# B&R Automation Studio project TD52 (part 138)

#### perm_par.var
```iecst
VAR
	pm_Error : UINT; (* permanent value error *) (* Deleted: pm : ParaMem_typ; permanent memory tags mathias, 22.8.11*)
	write_once : BOOL; (* write permanent memory once *)
	pm_len : UDINT; (* permanent value lenght *)
	ModuleName : STRING[35]; (* module name of object *)
	DatObjInfo_01 : DatObjInfo; (* data object info *)
	pm_id : UDINT; (* permanent value identifier *)
	pm_p : UDINT; (* permanent value pointer *)
	bCreateDataObj : BOOL; (* TRUE=create new data object *)
	perm_par_vers : UINT;
	DatObjRead_01 : DatObjRead; (* data object read *)
	usPMWriteCnt : UINT;
	DatObjDelete_PermMem : DatObjDelete;
	DatObjCreate_01 : DatObjCreate; (* data object create *)
	DatObjWrite_01 : DatObjWrite; (* data object write *)
	ulPMPointer : UDINT; (* adress of actual checksum value *)
	TON_WritePMEM : TON; (* delay write permanent memory *)
	ulChkValue : UDINT; (* actual value of parameter pointer *)
	bWriteDataObj : BOOL; (* TRUE=write data object module *)
	ulChecksum : UDINT; (* parameter checksum value *)
	ulChecksumOld : UDINT; (* last vlaue of parameter checksum *)
	TON_WarnDelay : TON;
END_VAR
VAR CONSTANT
	ERR_NOERROR : UINT := 0;
END_VAR
VAR
	tParaIntern : ParaHandler_typ; (*Connector type to perm_par*)
	xLocalParaCheck : ParaCheckFUB; (*local function instance to check parameter values*)
END_VAR
```

### Program Logical/ThermalReactor/VisTR (IEC) - Visualization

#### VisTRCyclic.st - Cyclic code
```iecst
(*******************************************************************************
VisTR	 			 Visualization signal to/from Thermal reactor module

This code is confidential AND proprietary to the INNIO Company.
It may NOT be used in any form, or reproduced in any manner,
without written permission of the INNIO Company.
Copyright, INNIO Company, 2019

Customized modifications: -
------------------------

History:
-------
V04.00.00	04-04-2014	Denk/Ganguly
V04.03.00	25-09-2014	Denk	Bugfix, OUT_TR.rP_ThR_EH / 1000;
									Adjust MM2VIS structure for VIS picture
V04.05.00	02-10-2017	Denk	Bugfix, MM2VIS.bThR_GT_COn1 and MM2VIS.bThR_GT_COn2 visibility with AND operation
V04.13.00	28-11-2023	Maran	Added auxiliary gas injection monitoring inputs
V04.14.00	27-11-2024	Maran	Added MM2VIS variables for el. heating status and auxiliary gas solenoid valve for ThR2

Instructions FOR use:
--------------------

Outstandings: -
------------

(*******************************************************************************)

PROGRAM _CYCLIC

	(* Module 2 VISU *)
	MM2VIS.b_ThR_Val_Air	:= OUT_TR.tThR_Val_Air.Do;
	MM2VIS.bThR_GT_COn1		:= OUT_TR.tThR_GT_COn1.Do AND OUT_TR.bThR_Val_SetOut;
	MM2VIS.bThR_GT_COn2		:= OUT_TR.tThR_GT_COn2.Do AND OUT_TR.bThR_Val_SetIn;
	MM2VIS.rP_ThR_EH		:= OUT_TR.rP_ThR_EH / 1000;
	MM2VIS.rT_ThR_Chamber	:= TK_moduleTR;
	MM2VIS.bThR_RelHeat		:= FG_HEIZG_moduleTR;
	MM2VIS.bThR_RelGas		:= OUT_TR.bThR_RelGas;
	MM2VIS.bThR_Val_SetIn	:= OUT_TR.bThR_Val_SetIn;
	MM2VIS.bThR_Val_SetOut	:= OUT_TR.bThR_Val_SetOut;

	IF Para.bThR2_Ena THEN //Thermal reactor 2
		// el. heating group - display of operating status for each of the five total groups
		IF OUT_TR.tThR2_EH_group1_Dem.Do	THEN	MM2VIS.iThR2_EH_group1_status := _iThR2_EH_Group_ON;
		ELSIF bThR2_EH_gr1_T_blocked		THEN	MM2VIS.iThR2_EH_group1_status := _iThR2_EH_Group_BLOCKED;
		ELSE MM2VIS.iThR2_EH_group1_status := _iThR2_EH_Group_OFF;
		END_IF
		IF OUT_TR.tThR2_EH_group2_Dem.Do	THEN	MM2VIS.iThR2_EH_group2_status := _iThR2_EH_Group_ON;
		ELSIF bThR2_EH_gr2_T_blocked		THEN	MM2VIS.iThR2_EH_group2_status := _iThR2_EH_Group_BLOCKED;
		ELSE MM2VIS.iThR2_EH_group2_status := _iThR2_EH_Group_OFF;
		END_IF
		IF OUT_TR.tThR2_EH_group3_Dem.Do	THEN	MM2VIS.iThR2_EH_group3_status := _iThR2_EH_Group_ON;
		ELSIF bThR2_EH_gr3_T_blocked		THEN	MM2VIS.iThR2_EH_group3_status := _iThR2_EH_Group_BLOCKED;
		ELSE MM2VIS.iThR2_EH_group3_status := _iThR2_EH_Group_OFF;
		END_IF
		IF OUT_TR.tThR2_EH_group4_Dem.Do	THEN	MM2VIS.iThR2_EH_group4_status := _iThR2_EH_Group_ON;
		ELSIF bThR2_EH_gr4_T_blocked		THEN	MM2VIS.iThR2_EH_group4_status := _iThR2_EH_Group_BLOCKED;
		ELSE MM2VIS.iThR2_EH_group4_status := _iThR2_EH_Group_OFF;
		END_IF
		IF OUT_TR.tThR2_EH_group5_Dem.Do	THEN	MM2VIS.iThR2_EH_group5_status := _iThR2_EH_Group_ON;
		ELSIF bThR2_EH_gr5_T_blocked		THEN	MM2VIS.iThR2_EH_group5_status := _iThR2_EH_Group_BLOCKED;
		ELSE MM2VIS.iThR2_EH_group5_status := _iThR2_EH_Group_OFF;
		END_IF

		// auxiliary gas solenoid valve - ThR2
		MM2VIS.bThR2_AuxGasShutOffValve_Dem := OUT_TR.tThR2_AuxGasShutOffValve_Dem.Do;
	END_IF
	(* from HalIO *)
	MM2VIS.rT_ThR_Chamber1_1		:= IN_TR.tT_ThR_Chamber1_1.Ai;
	MM2VIS.rT_ThR_Chamber1_2		:= IN_TR.tT_ThR_Chamber1_2.Ai;
	MM2VIS.rT_ThR_Chamber2_1		:= IN_TR.tT_ThR_Chamber2_1.Ai;
	MM2VIS.rT_ThR_Chamber2_2		:= IN_TR.tT_ThR_Chamber2_2.Ai;
	MM2VIS.rT_ThR_Comp				:= IN_TR.tT_ThR_Comp.Ai;
	MM2VIS.rT_ThR_In				:= IN_TR.tT_ThR_In.Ai;
	MM2VIS.rT_ThR_Out				:= IN_TR.tT_ThR_Out.Ai;
	MM2VIS.bPos_ThR_Val_In1			:= IN_TR.tPos_ThR_Val_In1.Di;
	MM2VIS.bPos_ThR_Val_In2			:= IN_TR.tPos_ThR_Val_In2.Di;
	MM2VIS.bPos_ThR_Val_Mid			:= IN_TR.tPos_ThR_Val_Mid.Di;
	MM2VIS.bPos_ThR_Val_Out1		:= IN_TR.tPos_ThR_Val_Out1.Di;
	MM2VIS.bPos_ThR_Val_Out2		:= IN_TR.tPos_ThR_Val_Out2.Di;
	MM2VIS.rPos_ThR_AuxGasCV_Act := IN_TR.tPos_ThR_AuxGasCV_Act.Ai;
	MM2VIS.rPr_ThR_AuxGasBeforeCV := IN_TR.tPr_ThR_AuxGasBeforeCV.Ai;
	MM2VIS.rPr_ThR_AuxGasAfterCV := IN_TR.tPr_ThR_AuxGasAfterCV.Ai;
	MM2VIS.rPr_ThR2_Inlet			:= IN_TR.tPr_ThR2_Inlet.Ai;
	MM2VIS.rPr_ThR2_Outlet			:= IN_TR.tPr_ThR2_Outlet.Ai;
	MM2VIS.rT_ThR2_LeftChamber		:= IN_TR.tT_ThR2_LeftChamber.Ai;
	MM2VIS.rT_ThR2_RightChamber		:= IN_TR.tT_ThR2_RightChamber.Ai;
	MM2VIS.rT_ThR2_Downstream		:= IN_TR.tT_ThR2_Downstream.Ai;
	MM2VIS.bThR2_T_fault_LeftCh		:= NOT IN_TR.tThR2_T_UnitOk_LeftCh.Di;
	MM2VIS.bThR2_T_fault_RightCh	:= NOT IN_TR.tThR2_T_UnitOk_RightCh.Di;
	MM2VIS.bThR2_T_fault_Downstream	:= NOT IN_TR.tThR2_T_UnitOk_Downstream.Di;
	MM2VIS.rT_ThR2_EH_group1		:= IN_TR.tT_ThR2_EH_group1.Ai;
	MM2VIS.rT_ThR2_EH_group2		:= IN_TR.tT_ThR2_EH_group2.Ai;
	MM2VIS.rT_ThR2_EH_group3		:= IN_TR.tT_ThR2_EH_group3.Ai;
	MM2VIS.rT_ThR2_EH_group4		:= IN_TR.tT_ThR2_EH_group4.Ai;
	MM2VIS.rT_ThR2_EH_group5		:= IN_TR.tT_ThR2_EH_group5.Ai;
	MM2VIS.bThR_LeftChamber_inlet	:= RM_KL_END_AUS;
	MM2VIS.bThR_RightChamber_inlet	:= RM_KL_END_EIN;

	(* VIS to module *)
	(*  ------  *)

	(* Controller *)
	tCtrTR_Heater_In			:= VIS2MM.tCtrTR_Heater_In;
	MM2VIS.tCtrTR_Heater_Out	:= tCtrTR_Heater_Out;

	(* For Debugging *)
	OUT_TR.rT_ThR_In			:= IN_TR.tT_ThR_In.Ai;
	OUT_TR.rT_ThR_Out			:= IN_TR.tT_ThR_Out.Ai;
	OUT_TR.rT_ThR_Chamber		:= TK_moduleTR;
	OUT_TR.rT_ThR_Chamber1_1	:= IN_TR.tT_ThR_Chamber1_1.Ai;
	OUT_TR.rT_ThR_Chamber1_2	:= IN_TR.tT_ThR_Chamber1_2.Ai;
	OUT_TR.rT_ThR_Chamber2_1	:= IN_TR.tT_ThR_Chamber2_1.Ai;
	OUT_TR.rT_ThR_Chamber2_2	:= IN_TR.tT_ThR_Chamber2_2.Ai;
	OUT_TR.rT_ThR_Comp			:= IN_TR.tT_ThR_Comp.Ai;

END_PROGRAM
```

#### VisTR.var - Local variables
```iecst
(********************************************************************
 * COPYRIGHT -- INNIO Company
 ********************************************************************
 * Program: VisTR
 * File: VisTR.var
 * Author: 105051626
 * Created: November 11, 2013
 ********************************************************************
 * Local variables of program VisTR
 ********************************************************************)

VAR

END_VAR

VAR CONSTANT
	_iThR2_EH_Group_ON : UINT := 2; (*Thermal reactor 2 - electrical heating group - status On*)
	_iThR2_EH_Group_OFF : UINT := 15; (*Thermal reactor 2 - electrical heating group - status Off*)
	_iThR2_EH_Group_BLOCKED : UINT := 42; (*Thermal reactor 2 - electrical heating group - status blocked*)
END_VAR
```

### Package Logical/Ventilation - VE: Ventilation

### Data object Logical/Ventilation/META_VE (Simple) - MODUL META data file

#### META_VE.dat
```
; *******************************************************************************
; AGGR: Module Meta Data (data module)
;
; This code is confidential and proprietary to the INNIO Company.
; It may not be used in any form, or reproduced in any manner, without the express
; written permission of the INNIO Company.
; Copyright, INNIO Company, 2022
;
; Customized modifications: -
; ------------------------
;
; History:
; -------
; V03.99.00.00	06.03.2013	Weitzer 	generated for modular software
;				02.10.2013	lettenb.	descriptions setted
;				04.12.2013	lettenb.	dependencies added
; V04.00.00.00	31.01.2014	lettenb.	version + dependencies changed
; V04.00.01.00	26.03.2014	lettenb.	version changed
; V04.00.03.00	22.07.2014	lettenb.	para_task update
; V04.03.00.00	02.03.2015	lettenb.	lockout warnings at plc cold restart
; V04.03.00.00	11.06.2015	Zengerer 	version + dependencies changed (IF change with array index 0 for compatibility with c-tasks)
;				15.06.2015  lettenb.	PARAMETER_CHK expanded
; V04.04.00.00	07.07.2015	lettenb.	version + dependencies changed
; 				20.03.2017	lettenb.	variant management room ventilation control, PID-contr.for engine room outlet fan regulation(temp.+pressure)
; V04.05.00.00	20.09.2017	Messner		Active Cooling Program added
;				22.12.2017	lettenb.	comment added: Safety-related application software source code (EN 13849-1 / 4.6.3)
; V04.05.01.00	01.03.2018	lettenb.	louver open/closed display, analog position added
; V04.06.00.00	16.07.2018	Perktold	2968 and 2969 Air inlet/outlet louver status signal failure added
; V04.07.00.00	09.08.2018	Schmid		change in tManAuxCtr struct (2nd low temperature charge cooling circuit)
;               29.10.2019  lettenb.	Vent_ER, man.aux.oper.mode for 1 lover bugfix, bu01
; V04.10.00.00	22.12.2020	lettenb.	config VAR.21/22: analog louvers with fix speed fans(set ZJAL1,ZJAL2,AJAL for this config.)(by jenbacher: not recommended config.)
; V04.11.00.00	23.11.2021	lettenb.	version changed
;				28.01.2022	Perktold	included plant controller upgrade
; V04.11.01.00	24.02.2022	Schmid		bAuxCust array size adjusted
; V04.12.00.00	07.12.2022	lettenb.	version changed
; V04.13.00.00	25.09.2023	Bacci		added IN_VE.tAuxV_Supply_Ok.Di in release FC
;				05.12.2023	Bacci		Added ventilation demand before starting the ingition selftest and exhaust scavenging. New DO for inlet louvers demand for customer (2023-190)
; V04.14.00.00	25.11.2024	Bacci		T6 Start procedure with purge start (2024-219): added ventilation demand before purge cranking cycle during fast start preparation
;				12.12.2024	Nagy		Room Ventilation Trip Redefinition (2024-226): added hi temperature warning and Louver alarm
; V4.25.00.00	26.11.2025	Bacci		Safety Function - Insufficient Ventilation (2024-202): reactivation of cold county function and safety plausibility check added
;
; Instructions for use:
; --------------------
; make only changes at the version numbers
;
; Outstandings:
; ------------
;
; *******************************************************************************
;
"<META>"
;
; Module ID
"<MODUL>VE</MODUL>"
;
; Module Version (xx.yy.zz.cc)
"<VERSION>04.25.00.00</VERSION>"
;
; Module Basisupdate Version BU (00-99)
"<BASISUPDATE_VERSION>00</BASISUPDATE_VERSION>"
;
; Optional: specify order number for limitated module usage
"<ORDER></ORDER>" ;<!--(optional for restricted customizations; missing statement makes module valid for all orders)-->
;
; Parameter Check <PARAn Name='aAbcdef' MIN='xxx' MAX='yyy' />  (watch for correct spacings and apostrophs!)
"<PARAMETER_CHK>"
"<PARA1 Name='iEng_Motortype' MIN='208' MAX='920' />"
"<PARA2 Name='rN_EngStart_LimHi' MIN='50.0' MAX='2200.0' />"
"<PARA3 />"
"<PARA4 />"
"<PARA5 />"
"</PARAMETER_CHK>"
;
; Permanent Datamodule Filenames<!-- NAME ist ohne Dateiendung einzutragen; Nur für Counter und interne Parameter verwenden-->
"<DATAMODULES>" ;<!-- optional; mehrere DATAMODULES erlaubt-->
"	<DATAMODULE>par_VE</DATAMODULE>"
"</DATAMODULES>"
;
; Dependencies Modules (MMxx.yy.zz.cc)
"<DEPENDENCIES>"
"	<DEPENDENCY MODULE='AB' VERSION='04.00.00.00' />"
"	<DEPENDENCY MODULE='AG' VERSION='04.14.00.00' />"
"	<DEPENDENCY MODULE='CH' VERSION='04.07.00.00' />"
"	<DEPENDENCY MODULE='CU' VERSION='04.07.00.00' />"
"	<DEPENDENCY MODULE='EC' VERSION='04.07.00.00' />"
"	<DEPENDENCY MODULE='EG' VERSION='04.25.00.00' />"
"	<DEPENDENCY MODULE='EX' VERSION='04.13.00.00' />"
"	<DEPENDENCY MODULE='GT' VERSION='04.00.00.00' />"
"	<DEPENDENCY MODULE='HA' VERSION='04.06.00.00' />"
"	<DEPENDENCY MODULE='HC' VERSION='04.07.00.00' />"
"	<DEPENDENCY MODULE='IG' VERSION='04.13.00.00' />"
"	<DEPENDENCY MODULE='OP' VERSION='04.03.00.00' />"
"	<DEPENDENCY MODULE='PB' VERSION='04.00.00.00' />"
"	<DEPENDENCY MODULE='SY' VERSION='04.03.00.00' />"
"   <DEPENDENCY VISVERSION='02.16.00.00' />"			; Dependencies Visualization
"</DEPENDENCIES>"
;
; Module function description
"<MODULEFUNCTION>" ;<!-- short overview documentation of module function; add reference to detailed information, if available-->
"	<General>	"
"	Control and monitoring engine room ventilation. "
"	</General>	"
""
"	<F1 Name='Engine room inlet temperature' LastModified='4.04.00.00'>"
"	Engine room inlet temperature monitoring.	"
"	</F1>"
"	<F2 Name='Engine room temperature' LastModified='4.04.00.00'>"
"	Engine room temperature monitoring and control.	"
"	</F2>"
"	<F3 Name='Engine room ventilation monitoring' LastModified='4.00.01.00'>"
"	Monitoring frequency converters, air flow sensor, doors.	"
"	</F3>"
"	<F4 Name='enter name of main function 3 here' LastModified='3.99.00.00'>"
"	Enter function 3 description for module here.	"
"	</F4>"
""
"	<Info>"
"   UPDATE V4.03.00	version + dependencies changed (IF change with array index 0 for compatibility with c-tasks)	"
"   UPDATE V4.07.00	change in tManAuxCtr struct	"
"	</Info>"
""
"	<Customized LastModified='3.99.00.00'>"
"	- Nothing "
"	</Customized>	"
""
"</MODULEFUNCTION>"
;
"</META>"
```

### module_VE.typ
```iecst
TYPE
	IN_Vent : 	STRUCT
		tAB2VE : AmmBase2MM;
		tPB2MM : ParaBase2MM_type;
		tERV_Op : HALioDi_Type; (*DI engine room ventilation operating/air flow ok*) (*OldName:DI_ERV_Op; Cycle:5;*)
		tERV_InlAir_Op : HALioDi_Type; (*DI engine room ventilation inlet-air operating/air flow ok*) (*OldName:newPv; Cycle:5;*)
		tERV_OutlAir_Op : HALioDi_Type; (*DI engine room ventilation outlet-air operating/air flow ok*) (*OldName:newPv; Cycle:5;*)
		tT_AirER_Ext_Hi1 : HALioDi_Type; (*DI room temperature limit *) (*OldName:RTM_25; Cycle:5;*)
		tT_AirER_Ext_Hi : HALioDi_Type; (*DI air engine room temperature external high*) (*OldName:RTM; Cycle:5;*)
		tT_AirER_Ext_Hi3 : HALioDi_Type; (*DI room temperature limit*) (*OldName:RTM_35; Cycle:5;*)
		tT_AirER_Ext_Hi2 : HALioDi_Type; (*DI room temperature limit*) (*OldName:RTM_30; Cycle:5;*)
		tER_Ext_Err : HALioDi_Type; (*DI engine room VE failure *) (*OldName:ST_RLV; Cycle:5;*)
		tER_InlAir_Ext_Err : HALioDi_Type; (*DI engine room inlet air VE failure *) (*OldName:ST_RLV; Cycle:5;*)
		tER_OutlAir_Ext_Err : HALioDi_Type; (*DI engine room outlet air VE failure *) (*OldName:ST_RLV; Cycle:5;*)
		tAirER_FS : HALioDi_Type; (*DI engine room VE flow switch*) (*OldName:DI_ERVent_FS; Cycle:5;*)
		tRel_ER_PurgeCycle : HALioDi_Type; (*DI release purge cycle*) (*OldName:DI_Rel_PurgeC; Cycle:5;*)
		tInAirER_Lou1Opened : HALioDi_Type; (*DI intake air engine room louver 1 open*) (*OldName:ZJAL1_O; Cycle:5;*)
		tInAirER_Lou2Opened : HALioDi_Type; (*DI intake air engine room louver 2 open*) (*OldName:ZJAL2_O; Cycle:5;*)
		tOutAirER_LouOpened : HALioDi_Type; (*DI outlet air engine room louver open*) (*OldName:AJAL_O; Cycle:5;*)
		tAuxV_Aux_ok : HALioDi_Type; (*DI auxiliary voltage supply ok Auxiliaries panel*) (*OldName:SPG_HBT; Cycle:5;*)
		tAuxV_ModIf_ok : HALioDi_Type; (*DI auxiliary voltage supply ok Module interface*) (*OldName:SPG_HBT; Cycle:5;*)
		tAuxV_Supply_Ok : HALioDi_Type; (*DI auxiliary voltage supply ok*) (*OldName:SPG_HBT; Cycle:5;*)
		tGCB_On : HALioDi_Type; (*DI generator circuit breaker closed*) (*OldName:GCB_ON; Cycle:5;*)
		rT_Ch_T1LP_Avg : REAL; (*average charge temperature before low-pressure turbocharger (= engine intake air) [°C]*) (*OldName:ssIATemp,ANA_ZLTP,tT_InAirER; Cycle:5;*) (* V04.04.00.00 *)
		bAMM_T_Ch_T1LP_Avg : BOOL; (*collective warning - average charge temp. before low-pressure TC (= engine intake air)*) (* V04.04.00.00 *)
		tT_AirER : HALioAi_Type; (*AI air engine room temperature [C]*) (*OldName:ANA_RTM; Cycle:5;*)
		rT_AirER_Customized : REAL; (*air engine room temperature customized [C]*) (*OldName:newPv; Cycle:5;*)
		tEng_Run : HALioDo_Type; (*Engine in operation*) (*OldName:M_BTRB; Cycle:5;*)
		tPos_InlLou1 : HALioAi_Type; (*AI position air inlet louver 1 [%]*) (*OldName:newPv; Cycle:5;*) (*STM*)
		tPos_InlLou2 : HALioAi_Type; (*AI position air inlet louver 2 [%]*) (*OldName:newPv; Cycle:5;*) (*STM*)
		rPos_InlLou1 : REAL; (*position air inlet louver 1 [%]*) (*OldName:newPv; Cycle:5;*) (*STM*)
		rPos_InlLou2 : REAL; (*position air inlet louver 2 [%]*) (*OldName:newPv; Cycle:5;*) (*STM*)
		tPos_OutlLou1 : HALioAi_Type; (*AI position air outlet louver 1 [%]*) (*OldName:newPv; Cycle:5;*) (*STM*)
		tPos_OutlLou2 : HALioAi_Type; (*AI position air outlet louver 2 [%]*) (*OldName:newPv; Cycle:5;*) (*STM*)
		rPos_OutlLou1 : REAL; (*position air outlet louver 1 [%]*) (*OldName:newPv; Cycle:5;*) (*STM*)
		rPos_OutlLou2 : REAL; (*position air outlet louver 2 [%]*) (*OldName:newPv; Cycle:5;*) (*STM*)
		tPos_CircLou1 : HALioAi_Type; (*AI position air circulation louver 1 [%]*) (*OldName:newPv; Cycle:5;*) (*STM*)
		tPos_CircLou2 : HALioAi_Type; (*AI position air circulation louver 2 [%]*) (*OldName:newPv; Cycle:5;*) (*STM*)
		rPos_CircLou1 : REAL; (*position air circulation louver 1 [%]*) (*OldName:newPv; Cycle:5;*) (*STM*)
		rPos_CircLou2 : REAL; (*position air circulation louver 2 [%]*) (*OldName:newPv; Cycle:5;*) (*STM*)
		tPrDiff_ER : HALioAi_Type; (*AI engine room difference pressure [mbar]*) (*OldName:newPv; Cycle:5;*) (*STM 2*)
		rPrDiff_ER : REAL; (*engine room difference pressure [mbar]*) (*OldName:newPv; Cycle:5;*) (*STM 2*)
		bMsg1031 : BOOL; (*Alarm 1031 Emergency stop*) (*OldName:M_SIS; Cycle:5;*)
		bMsg1052 : BOOL; (*Alarm 1052 gas prealarm*) (*OldName:M_GALV; Cycle:5;*)
		bMsg1053 : BOOL; (*Alarm 1053 Gas Alarm*) (*OldName:M_GAL; Cycle:5;*)
		bMsg1054 : BOOL; (*Alarm 1054 Fire alarm*) (*OldName:M_BAL; Cycle:5;*)
		bMsg3003 : BOOL; (*3003 Measurement signal disturbance*) (*OldName:M_MS; Cycle:5;*)
		bEng_Aux_Dem_CDR : BOOL; (*engine auxiliaries demand with cool down run*) (*OldName:ANFHBT; Cycle:5;*)
		bEng_Dem_EPS : BOOL; (*Engine demand for emergency operation*) (*OldName:M_NANF; Cycle:5;*)
		bOnly_Island : BOOL; (*only island operation*) (*OldName:REIN_INSEL; Cycle:5;*)
		bRel_ScavN2 : BOOL; (*conditions for scavenge with N2*) (*OldName:FG_N2; Cycle:5;*)
		iSt_OpMode : UDINT; (*engine operating mode*) (*OldName:newPv; Cycle:5;*)
		bEng_Dem : BOOL; (*module demanded*) (*OldName:M_AGFD; Cycle:5;*)
		bGV_On : BOOL; (*command open gas valves*) (*OldName:M_GASV; Cycle:5;*)
		bEng_Aux_Dem : BOOL; (*engine auxiliaries demand*) (*OldName:M_ANFHBT; Cycle:5;*)
		iIdx_OMSS : INT; (*engine operating mode selection*) (*OldName:newPv; Cycle:5;*)
		bInAirER_FanSet100 : BOOL; (*demand engine room fan 100% speed*) (*OldName:LUE100; Cycle:5;*)
		rP_Act_Norm_Filt : REAL; (*Actual power related to rP_Nom filtered T=1s [%/P_Nom]*) (*OldName:P_IST; Cycle:5;*)
		rN_EngAct : REAL; (* engine speed actual [1/min] *) (*OldName:n_ist; Cycle:5*)
		tER_DoorClosed : HALioDi_Type; (*DI engine room doors closed*) (*OldName:DI_ER_DoorClosed; Cycle:5;*)
		rCust_SparePara : ARRAY[0..200]OF REAL; (*SPS_REZP1 to SPS_REZP200	*) (* OldName: SPS_REZP1, SPS_REZP2, SPS_REZP70; Cycle: 5; *)
		tCustAnaIn : ARRAY[0..120]OF HALioAi_Type; (*Replacement for RAN_KANAL...*) (*OldName: ANA_RAN	; Cycle: 5;*)
		tCustDigIn : ARRAY[0..200]OF HALioDi_Type; (*new, reserved for Project specific use*) (*OldName: new PV	; Cycle: 5;*)
		tManAuxCtr : tManAuxCtr_typ; (*Manual operating auxiliaries control - Handbedienebene*) (*OldName: new PV; Cycle: 5;*)
		tDPr_InAirFiltERV_Hi : HALioDi_Type; (*air inlet filter difference pressure high - engine room ventilation*) (*OldName: E_FILTER; Cycle: 5;*)
		tFireProtFlap1_InlAir_Closed : HALioDi_Type; (*fireprotectionflap 1 inlet-air closed*) (*OldName:newPv; Cycle:5;*)
		tFireProtFlap2_InlAir_Closed : HALioDi_Type; (*fireprotectionflap 2 inlet-air closed*) (*OldName:newPv; Cycle:5;*)
		tFireProtFlap1_InlAir_Opened : HALioDi_Type; (*fireprotectionflap 1 inlet-air opened*) (*OldName:newPv; Cycle:5;*)
		tFireProtFlap2_InlAir_Opened : HALioDi_Type; (*fireprotectionflap 2 inlet-air opened*) (*OldName:newPv; Cycle:5;*)
		tFireProtFlap1_OutlAir_Closed : HALioDi_Type; (*fireprotectionflap 1 outlet-air closed*) (*OldName:newPv; Cycle:5;*)
		tFireProtFlap2_OutlAir_Closed : HALioDi_Type; (*fireprotectionflap 2 outlet-air closed*) (*OldName:newPv; Cycle:5;*)
		tFireProtFlap1_OutlAir_Opened : HALioDi_Type; (*fireprotectionflap 1 outlet-air opened*) (*OldName:newPv; Cycle:5;*)
		tFireProtFlap2_OutlAir_Opened : HALioDi_Type; (*fireprotectionflap 2 outlet-air opened*) (*OldName:newPv; Cycle:5;*)
		bFS_Act : BOOL; (*FastStart activated (enabled and required from customer)*) (*Oldname:new PV, Cycle:5*)
		bACP_AirER_Dem : BOOL; (* Active Cooling Program Room Air Ventilation demanded *) (*OldName:newPv; Cycle:5;*)
		tInAirER_Lou1Closed : HALioDi_Type; (*DI intake air engine room louver 1 Closed*)
		tInAirER_Lou2Closed : HALioDi_Type; (*DI intake air engine room louver 2 Closed*)
		tOutAirER_LouClosed : HALioDi_Type; (*DI outlet air engine room louver Closed*)
		bInLouDemIgn : BOOL; (*Inlet louver demand for ignition selftest*)
		bInLouDemEX : BOOL; (*Inlet louver demand for scavenging*)
		bInLouDemAG : BOOL; (*Inlet louver demand for purge cranking cycle for fast start*)
		bERV_PC_Forced : BOOL; (*SAFETY PLC: Force ERV safety plausibility checks*)
		bSafetyPLC_Active : BOOL; (*SAFETY PLC: SafetyPLC is active*) (*OldName: new PV; Cycle: 5;*)
	END_STRUCT;
	OUT_Vent : 	STRUCT
		tVE2AB : MM2AmmBase;
		tVE2PB : MM2ParaBase_type;
		tRel_ER_Fan : HALioDo_Type; (*DO demand VE > min. speed*) (*OldName:FG_LUE; Cycle:5;*)
		tSet_ER_Fan_Min : HALioDo_Type; (*DO demand VE min. speed*) (*OldName:LUE_MIN; Cycle:5;*)
		tDemPurgeER : HALioDo_Type; (*DO demand room VE for purge cycle*) (*OldName:DO_DmndPurge; Cycle:5;*)
		tRel_ER_FC : HALioDo_Type; (*DO release frequency converter for room VE*) (*OldName:FG_FU; Cycle:5;*)
		tInAirER_Fan1DemOn : HALioDo_Type; (*DO demand air inlet ventilator 1*) (*OldName:ZLVST_1; Cycle:5;*)
		tInAirER_Fan2DemOn : HALioDo_Type; (*DO demand air inlet ventilator 2*) (*OldName:ZLVST_2; Cycle:5;*)
		tOutAirER_LouDemOpen : HALioDo_Type; (*DO demand open air outlet louver *) (*OldName:A_AJAL; Cycle:5;*)
		tInAirER_Lou2DemOpen : HALioDo_Type; (*DO demand open air inlet louver 2*) (*OldName:A_ZJAL2; Cycle:5;*)
		tInAirER_Lou1DemOpen : HALioDo_Type; (*DO demand open air inlet louver 1*) (*OldName:A_ZJAL1; Cycle:5;*)
		tCtr_InlLou_Set : HALioAo_Type; (*AO inlet-air louver setpoint*) (*OldName:newPv; Cycle:5;*) (*STM*)
		tCtr_OutlLou_RT_Set : HALioAo_Type; (*AO outlet-air louver setpoint regarding engine room temperature*) (*OldName:newPv; Cycle:5;*) (*STM 2*)
		tCtr_OutlLou_RDP_Set : HALioAo_Type; (*AO outlet-air louver setpoint regarding engine room differential pressure*) (*OldName:newPv; Cycle:5;*) (*STM 2*)
		tCtr_CircLou_Set : HALioAo_Type; (*AO circulation-air louver setpoint*) (*OldName:newPv; Cycle:5;*) (*STM*)
		tER_FC_Set : HALioAo_Type; (*AO engine room frequency converter setpoint [%]*) (*OldName:REG12_y; Cycle:5;*)
		bMsg2295 : BOOL; (*engine room ventilation failure inlet air*) (*OldName:newPv; Cycle:5;*)
		bMsg2296 : BOOL; (*engine room ventilation failure outlet air*) (*OldName:newPv; Cycle:5;*)
		bMsg2701 : BOOL; (*position air inlet louver 1 signal failure*) (*OldName:newPv; Cycle:5;*) (*STM*)
		bMsg2702 : BOOL; (*position air inlet louver 2 signal failure*) (*OldName:newPv; Cycle:5;*) (*STM*)
		bMsg2703 : BOOL; (*position air outlet louver 1 signal failure*) (*OldName:newPv; Cycle:5;*) (*STM*)
		bMsg2704 : BOOL; (*position air outlet louver 2 signal failure*) (*OldName:newPv; Cycle:5;*) (*STM*)
		bMsg2705 : BOOL; (*engine room difference pressure signal failure*) (*OldName:newPv; Cycle:5;*) (*STM*)
		bMsg2706 : BOOL; (*engine room difference pressure low*) (*OldName:newPv; Cycle:5;*) (*STM*)
		bMsg2707 : BOOL; (*engine room difference pressure high*) (*OldName:newPv; Cycle:5;*) (*STM*)
		bMsg2708 : BOOL; (*position air circulation louver 1 signal failure*) (*OldName:newPv; Cycle:5;*) (*STM*)
		bMsg2709 : BOOL; (*position air circulation louver 2 signal failure*) (*OldName:newPv; Cycle:5;*) (*STM*)
		bMsg2795 : BOOL; (*engine room ventilation failure inlet air*) (*OldName:newPv; Cycle:5;*)
		bMsg2796 : BOOL; (*engine room ventilation failure outlet air*) (*OldName:newPv; Cycle:5;*)
		bMsg2797 : BOOL; (*parameterization error air inlet louvers*) (*OldName:newPv; Cycle:5;*)
		bMsg2798 : BOOL; (*parameterization error air outlet louvers*) (*OldName:newPv; Cycle:5;*)
		bMsg3152 : BOOL; (*engine room temperature signal failure*) (*OldName:M_MSRTM_W; Cycle:5;*)
		bPurgeER_Rdy : BOOL; (*purge cycle ready*) (*OldName:purge_rdy; Cycle:5;*)
		rP_Red_T_InAirER_Norm : REAL; (*power reduction by engine room air inlet temperature [%]*) (*OldName:newPv; Cycle:5;*)
		tCtr_OutlVE_RT_Set : HALioAo_Type; (*AO outlet-air ventilation setpoint regarding engine room temperature*) (*OldName:newPv; Cycle:5;*)
		tCtr_OutlVE_RDP_Set : HALioAo_Type; (*AO outlet-air ventilation setpoint regarding engine room differential pressure*) (*OldName:newPv; Cycle:5;*)
		Pos_OutlLou2_OK : BOOL; (*position feedback air outlet louver 2 OK depending on parameter*)
		Pos_OutlLou1_OK : BOOL; (*position feedback air outlet louver 1 OK depending on parameter*)
		Pos_InlLou2_OK : BOOL; (*position feedback air inlet louver 2 OK depending on parameter*)
		Pos_InlLou1_OK : BOOL; (*position feedback air inlet louver 1 OK depending on parameter*)
		bERV_NotRdy : BOOL; (*engine room ventilation not ready - block engine start*)
		tInAirER_Lou1Opened : HALioDi_Type; (*DI intake air engine room louver 1 open*)
		tInAirER_Lou2Opened : HALioDi_Type; (*DI intake air engine room louver 2 open*)
		tOutAirER_LouOpened : HALioDi_Type; (*DI outlet air engine room louver open*)
		tDemERVentInLou_Cust : HALioDo_Type; (*DO inlet louvers demand for customer*)
		bInLouRelVE : BOOL; (*inlet louvers open or not closed*)
		bERV_ColdCountry : BOOL; (*SAFETY PLC: Cold country mode active for safety PLC*)
		bERV_Lou_PC_OP : BOOL; (*SAFETY PLC: Plausibility check for opening the louvres*)
		bERV_Lou_PC_CL : BOOL; (*SAFETY PLC: Plausibility check for closing the louvres*)
	END_STRUCT;
	VIS2MM_Struct : 	STRUCT
		tCtr_InlLou_In : _tGeACtrIn; (*inlet-air louver controller (for engine room temperature)*) (*OldName:newPv; Cycle:5;*) (*STM*)
		tCtr_OutlLou_RT_In : _tGeACtrIn; (*outlet-air louver controller (for engine room temperature)*) (*OldName:newPv; Cycle:5;*) (*STM 2*)
		tCtr_OutlVE_RT_In : _tGeACtrIn; (*outlet-air ventilation controller (for engine room temperature)*) (*OldName:newPv; Cycle:5;*)
		tCtr_OutlLou_RDP_In : _tGeACtrIn; (*outlet-air louver controller (for engine room differential pressure)*) (*OldName:newPv; Cycle:5;*) (*STM 2*)
		tCtr_OutlVE_RDP_In : _tGeACtrIn; (*outlet-air ventilation controller (for engine room differential pressure)*) (*OldName:newPv; Cycle:5;*)
		tCtr_CircLou_In : _tGeACtrIn; (*circulation-air louver controller (for intake air temperature)*) (*OldName:newPv; Cycle:5;*) (*STM*)
		tCtr_ER_In : _tGeACtrIn; (*engine room temperature controller*) (*OldName:REG12; Cycle:5;*)
	END_STRUCT;
	MM2VIS_Struct : 	STRUCT
		tCtr_InlLou_Out : _tGeACtrOut; (*inlet-air louver controller (for engine room temperature)*) (*OldName:newPv; Cycle:5;*) (*STM*)
		tCtr_OutlLou_RT_Out : _tGeACtrOut; (*outlet-air louver controller (for engine room temperature)*) (*OldName:newPv; Cycle:5;*) (*STM 2*)
		tCtr_OutlVE_RT_Out : _tGeACtrOut; (*outlet-air ventilation controller (for engine room temperature)*) (*OldName:newPv; Cycle:5;*)
		tCtr_OutlLou_RDP_Out : _tGeACtrOut; (*outlet-air louver controller (for engine room differential pressure)*) (*OldName:newPv; Cycle:5;*) (*STM 2*)
		tCtr_OutlVE_RDP_Out : _tGeACtrOut; (*outlet-air ventilation controller (for engine room differential pressure)*) (*OldName:newPv; Cycle:5;*)
		tCtr_CircLou_Out : _tGeACtrOut; (*circulation-air louver controller (for intake air temperature)*) (*OldName:newPv; Cycle:5;*) (*STM*)
		tCtr_ER_Out : _tGeACtrOut; (*engine room temperature controller*) (*OldName:REG12; Cycle:5;*)
		rCtr_OutlVE_RDP_Set : REAL; (*vis speed setpoint outlet ventilation [%]*)
		rT_AirER : REAL; (*vis air engine room temperature [°C]*) (*OldName:ANA_RTM; Cycle:5;*)
		rPrDiff_ER : REAL; (*vis engine room difference pressure [mbar]*) (*OldName:newPv; Cycle:5;*) (*STM 2*)
		rP_Red_T_InAirER_Norm : REAL; (*power reduction by engine room inlet air temperature [%]*) (*OldName:newPv; Cycle:5;*)
		rPos_InlLou1 : REAL; (*position air inlet louver 1 [%]*) (*OldName:newPv; Cycle:5;*) (*STM*)
		rPos_InlLou2 : REAL; (*position air inlet louver 2 [%]*) (*OldName:newPv; Cycle:5;*) (*STM*)
		rPos_OutlLou1 : REAL; (*position air outlet louver 1 [%]*) (*OldName:newPv; Cycle:5;*) (*STM*)
		rPos_OutlLou2 : REAL; (*position air outlet louver 2 [%]*) (*OldName:newPv; Cycle:5;*) (*STM*)
		rPos_CircLou1 : REAL; (*position air circulation louver 1 [%]*) (*OldName:newPv; Cycle:5;*) (*STM*)
		rPos_CircLou2 : REAL; (*position air circulation louver 2 [%]*) (*OldName:newPv; Cycle:5;*) (*STM*)
		bInAirER_Lou1Opened : BOOL; (*vis inlet air engine room louver 1 opened*) (*OldName:B_SV[33]; Cycle:5;*)
		bInAirER_Lou2Opened : BOOL; (*vis inlet air engine room louver 2 opened*) (*OldName:B_SV[34]; Cycle:5;*)
		bOutAirER_LouOpened : BOOL; (*vis outlet air engine room louver opened*) (*OldName:B_SV[35]; Cycle:5;*)
		bInAirER_Fan1DemOn : BOOL; (*vis demand air inlet ventilator 1*) (*OldName:B_SV[36]; Cycle:5;*)
		bInAirER_Fan2DemOn : BOOL; (*vis demand air inlet ventilator 2*) (*OldName:B_SV[37]; Cycle:5;*)
		bInAirER_FanSet100 : BOOL; (*vis demand engine room fan 100% speed*) (*OldName:LUE100; Cycle:5;*)
		bRel_ER_Fan : BOOL; (*engine room fan release*) (*OldName:FG_FU; Cycle:5;*)
		bFireProtFlap1_InlAir_Opened : BOOL; (*vis status fire protection flap 1 inlet air *) (*OldName:newPv; Cycle:5;*)
		bFireProtFlap2_InlAir_Opened : BOOL; (*vis status fire protection flap 2 inlet air *) (*OldName:newPv; Cycle:5;*)
		bFireProtFlap1_OutlAir_Opened : BOOL; (*vis status fire protection flap 1 outlet air *) (*OldName:newPv; Cycle:5;*)
		bFireProtFlap2_OutlAir_Opened : BOOL; (*vis status fire protection flap 2 outlet air *) (*OldName:newPv; Cycle:5;*)
		bCtrER_YFix : BOOL; (*demand engine room controller activation with fixed y*)
		bMsg1135 : BOOL; (*air engine room temperature high*) (*OldName:AMM_Axxxx[]; Cycle:5;*)
		bMsg1138 : BOOL; (*engine room fan failure trip*) (*OldName:AMM_Axxxx[]; Cycle:5;*)
		bMsg2120 : BOOL; (*engine room fan failure*) (*OldName:AMM_Wxxxx[]; Cycle:5;*)
		bMsg2295 : BOOL; (*engine room ventilation failure inlet air*) (*OldName:newPv; Cycle:5;*)
		bMsg2296 : BOOL; (*engine room ventilation failure outlet air*) (*OldName:newPv; Cycle:5;*)
		bMsg2630 : BOOL; (*difference pressure filter high - engine room ventilation*) (*OldName:newPv; Cycle:5;*)
		bMsg2701 : BOOL; (*position air inlet louver 1 signal failure*) (*OldName:newPv; Cycle:5;*) (*STM*)
		bMsg2702 : BOOL; (*position air inlet louver 2 signal failure*) (*OldName:newPv; Cycle:5;*) (*STM*)
		bMsg2703 : BOOL; (*position air outlet louver 1 signal failure*) (*OldName:newPv; Cycle:5;*) (*STM*)
		bMsg2704 : BOOL; (*position air outlet louver 2 signal failure*) (*OldName:newPv; Cycle:5;*) (*STM*)
		bMsg2705 : BOOL; (*engine room difference pressure signal failure*) (*OldName:newPv; Cycle:5;*) (*STM*)
		bMsg2706 : BOOL; (*engine room difference pressure low*) (*OldName:newPv; Cycle:5;*) (*STM*)
		bMsg2707 : BOOL; (*engine room difference pressure high*) (*OldName:newPv; Cycle:5;*) (*STM*)
		bMsg2708 : BOOL; (*position air circulation louver 1 signal failure*) (*OldName:newPv; Cycle:5;*) (*STM*)
		bMsg2709 : BOOL; (*position air circulation louver 2 signal failure*) (*OldName:newPv; Cycle:5;*) (*STM*)
		bMsg2795 : BOOL; (*engine room ventilation failure inlet air*) (*OldName:newPv; Cycle:5;*)
		bMsg2796 : BOOL; (*engine room ventilation failure outlet air*) (*OldName:newPv; Cycle:5;*)
		bMsg2797 : BOOL; (*parameterization error air inlet louvers*) (*OldName:newPv; Cycle:5;*)
		bMsg2798 : BOOL; (*parameterization error air outlet louvers*) (*OldName:newPv; Cycle:5;*)
		bMsg3152 : BOOL; (*engine room air temperature signal failure*) (*OldName:AMM_Wxxxx[]; Cycle:5;*)
		bMsg3223 : BOOL; (*engine room air inlet temperature signal failure*) (*OldName:AMM_Wxxxx[]; Cycle:5;*)
		bMsg3224 : BOOL; (*engine room air inlet temperature high*) (*OldName:AMM_Wxxxx[]; Cycle:5;*)
		bMsg3302 : BOOL; (*purge cycle incomplete*) (*OldName:AMM_Axxxx[]; Cycle:5;*)
		bMsg3367 : BOOL; (*engine room ventilation failure - doors*) (*OldName:AMM_Axxxx[]; Cycle:5;*)
		bMsg3571 : BOOL; (*no release start module from purge cycle*) (*OldName:AMM_Wxxxx[]; Cycle:5;*)
		bMsg2968 : BOOL; (*Air inlet louver status signal failure*)
		bMsg2969 : BOOL; (*Air outlet louver status signal failure*)
		bMsg2472 : BOOL; (*Room temperature high warning*)
		bMsg9401 : BOOL; (*Louvers failure*)
	END_STRUCT;
	tManAuxCtr_typ : 	STRUCT
		bGnl_Rel : BOOL; (*General release. Safety conditions (gas alarm, fire alarm, safety loop, ..) are OK.*) (*OldName: new PV; Cycle: 5;*)
		bECWP_PreH_COf_Man : BOOL; (*engine cooling water pump preheating demand off*) (*OldName: new PV; Cycle: 5;*)
		bECW_PreH_COf_Man : BOOL; (*engine cooling water preheating demand off*) (*OldName: new PV; Cycle: 5;*)
		bInAirER_Lou2DemOpen_Man : BOOL; (*demand open air inlet louver 2*) (*OldName: new PV; Cycle:5;*)
		bInAirER_Lou1DemOpen_Man : BOOL; (*demand open air inlet louver 1*) (*OldName: new PV; Cycle:5;*)
		bOutAirER_LouDemOpen_Man : BOOL; (*open air outlet louver *) (*OldName: new PV; Cycle:5;*)
		bInAirER_Fan1DemOn_Man : BOOL; (*demand air inlet ventilator 1*) (*OldName: new PV; Cycle:5;*)
		bInAirER_Fan2DemOn_Man : BOOL; (*demand air inlet ventilator 2*) (*OldName: new PV; Cycle:5;*)
		bER_FC_Set_Man : BOOL; (*demand engine room frequency converter setpoint*) (*OldName: new PV; Cycle:5;*)
		rER_FC_Set_Man : REAL; (*engine room frequency converter setpoint [%]*) (*OldName: new PV; Cycle:5;*)
		bER_OutlV_FC_Set_Man : BOOL; (*demand engine room air outlet ventilation frequency converter setpoint*) (*OldName: new PV; Cycle:5;*)
		rER_OutlV_FC_Set_Man : REAL; (*engine room air outlet ventilation frequency converter setpoint [%]*) (*OldName: new PV; Cycle:5;*)
		bEC_DemPump_Man : BOOL; (*emergency cooler demand pump*) (*OldName: new PV; Cycle:5;*)
		bEC_DemFan_Man : BOOL; (*emergency cooler demand fan 1 - 16*) (*OldName: new PV; Cycle:5;*)
		bChC_DemPump_Man : BOOL; (*charge cooler demand pump*) (*OldName: new PV; Cycle:5;*)
		bChC_DemFan_Man : BOOL; (*charge cooler demand fan 1 - 16*) (*OldName: new PV; Cycle:5;*)
		bEG_BoVaCoOpen_Man : BOOL; (*exhaust gas boiler valve command open*) (*OldName: new PV; Cycle:5;*)
		bEG_BoVaCoClose_Man : BOOL; (*exhaust gas boiler valve command close*) (*OldName: new PV; Cycle:5;*)
		bEG_ByVaCoOpen_Man : BOOL; (*exhaust gas bypass valve command open*) (*OldName: new PV; Cycle:5;*)
		bEG_ByVaCoClose_Man : BOOL; (*exhaust gas bypass valve command close*) (*OldName: new PV; Cycle:5;*)
		bAuxCust_Man : ARRAY[0..40]OF BOOL; (*reserve customer auxiliaries*) (*OldName: new PV; Cycle:5;*)
		bCDP_Dem_Man : BOOL; (*demand condensor pump*) (*OldName: new PV; Cycle:5;*)
		bBHV_Dem_Man : BOOL; (*demand boiler house ventilation*) (*OldName: newPv; Cycle:5;*)
		bHWF_Dem_Man : BOOL; (*demand heating circuit flap*) (*OldName:newPv; Cycle:5;*)
		bChC_Heating_Man : BOOL; (*charge cooler pre heating*) (*OldName:newPv; Cycle:5;*)
		bCO2_DemCodinox_Man : BOOL; (*CO2 demand CODINOX*) (*OldName:newPv; Cycle:5;*)
		bECWP_PreH_COf : BOOL; (*engine cooling water pump preheating demand off*) (*OldName: new PV; Cycle: 5;*)
		bECW_PreH_COf : BOOL; (*engine cooling water preheating demand off*) (*OldName: new PV; Cycle: 5;*)
		bInAirER_Lou2DemOpen : BOOL; (*demand open air inlet louver 2*) (*OldName: new PV; Cycle:5;*)
		bInAirER_Lou1DemOpen : BOOL; (*demand open air inlet louver 1*) (*OldName: new PV; Cycle:5;*)
		bOutAirER_LouDemOpen : BOOL; (*open air outlet louver *) (*OldName: new PV; Cycle:5;*)
		bInAirER_Fan1DemOn : BOOL; (*demand air inlet ventilator 1*) (*OldName: new PV; Cycle:5;*)
		bInAirER_Fan2DemOn : BOOL; (*demand air inlet ventilator 2*) (*OldName: new PV; Cycle:5;*)
		bER_OutlV_FC_Set : BOOL; (*demand engine room air outlet ventilation frequency converter setpoint*) (*OldName: new PV; Cycle:5;*)
		rER_OutlV_FC_Set : REAL; (*engine room air outlet ventilation frequency converter setpoint [%]*) (*OldName: new PV; Cycle:5;*)
		bER_FC_Set : BOOL; (*demand engine room frequency converter setpoint*) (*OldName: new PV; Cycle:5;*)
		rER_FC_Set : REAL; (*engine room frequency converter setpoint [%]*) (*OldName: new PV; Cycle:5;*)
		bEC_DemPump : BOOL; (*emergency cooler demand pump*) (*OldName: new PV; Cycle:5;*)
		bEC_DemFan : BOOL; (*emergency cooler demand fan 1 - 16*) (*OldName: new PV; Cycle:5;*)
		bChC_DemPump : BOOL; (*charge cooler demand pump*) (*OldName: new PV; Cycle:5;*)
		bChC_DemFan : BOOL; (*charge cooler demand fan 1 - 16*) (*OldName: new PV; Cycle:5;*)
		bEG_BoVaCoOpen : BOOL; (*exhaust gas boiler valve command open*) (*OldName: new PV; Cycle:5;*)
		bEG_BoVaCoClose : BOOL; (*exhaust gas boiler valve command close*) (*OldName: new PV; Cycle:5;*)
		bEG_ByVaCoOpen : BOOL; (*exhaust gas bypass valve command open*) (*OldName: new PV; Cycle:5;*)
		bEG_ByVaCoClose : BOOL; (*exhaust gas bypass valve command close*) (*OldName: new PV; Cycle:5;*)
		bAuxCust : ARRAY[0..70]OF BOOL; (*reserve customer auxiliaries*) (*OldName: new PV; Cycle:5;*)
		bCDP_Dem : BOOL; (*demand condensor pump*) (*OldName: new PV; Cycle:5;*)
		bBHV_Dem : BOOL; (*demand boiler house ventilation*) (*OldName: newPv; Cycle:5;*)
		bHWF_Dem : BOOL; (*demand heating circuit flap*) (*OldName:newPv; Cycle:5;*)
		bChC_Heating : BOOL; (*charge cooler pre heating*) (*OldName:newPv; Cycle:5;*)
		bCO2_DemCodinox : BOOL; (*CO2 demand CODINOX*) (*OldName:newPv; Cycle:5;*)
		bChC2_DemPump : BOOL; (*charge cooler 2 demand pump*) (*OldName: new PV; Cycle:5;*)
		bChC2_DemPump_Man : BOOL; (*charge cooler 2 demand pump*) (*OldName: new PV; Cycle:5;*)
		bChC2_DemFan : BOOL; (*charge cooler 2 demand fan 1 - 16*) (*OldName: new PV; Cycle:5;*)
		bChC2_DemFan_Man : BOOL; (*charge cooler 2 demand fan 1 - 16*) (*OldName: new PV; Cycle:5;*)
		bChC2_Heating : BOOL; (*charge cooler 2 pre heating*) (*OldName:newPv; Cycle:5;*)
		bChC2_Heating_Man : BOOL; (*charge cooler 2 pre heating*) (*OldName:newPv; Cycle:5;*)
		bECW_HydrPreH_COf : BOOL; (*engine cooling water hydraulic preheating demand off*) (*OldName: new PV; Cycle: 5;*)
		bECW_HydrPreH_COf_Man : BOOL; (*engine cooling water hydraulic preheating demand off*) (*OldName: new PV; Cycle: 5;*)
		bEOP_DemPump : BOOL; (*engine prelubrication pump manual demand*) (*OldName: new PV; Cycle: 5;*)
		bEOP_DemPump_Man : BOOL; (*engine prelubrication pump manual demand*) (*OldName: new PV; Cycle: 5;*)
	END_STRUCT;
END_TYPE
```

### module_VEPara.typ
```iecst
TYPE
	PROGRAMMER_INFO : 	STRUCT
		DO_NOT_SORT_PARA : STRING[40] := 'DO NOT CHANGE PARAMETER SORTING!'; (*DO NOT CHANGE PARAMETER SORTING!*) (*ADD NEW PARAMETER ONLY AT THE END OF THE Para STRUCTURE. DO NOT DELETE existing Para items.*)
	END_STRUCT;
	Para_Vent : 	STRUCT
		tCtr_ER : _tGeACtrPara; (*Para controller engine room temperature*) (*OldName:REG12; Cycle:5;*)
		bCtr_ER : BOOL; (*PARA [12245]: engine room ventilation controller enable*) (*OldName:bPlantCtr12; Cycle:5;*)
		bAuxER_Vent_Visible : BOOL; (*PARA [12244]: auxiliaries engine room ventilation visible*) (*OldName:bAuxilAirVent; Cycle:5;*)
		iEng_Motortype : INT; (*Para motortype*) (*OldName:motortyp; Cycle:5;*)
		bVISA : BOOL; (*PARA [12259]: monitoring according VISA*) (*OldName:newPv; Cycle:5;*)
		bLouvers : BOOL; (*PARA [12253]: engine room ventilation with louvers*) (*OldName:newPv; Cycle:5;*)
		bER_VentColdCountryMode : BOOL; (*PARA [12246]: engine room VE cold country mode*) (*OldName:newPv; Cycle:5;*)
		rT_CtrER_WexStop : REAL; (*PARA [12272]: engine room temperature controller external setpoint stop*) (*OldName:W2_RTMREG; Cycle:5;*)
		rT_CtrER_WexRun : REAL; (*PARA [12271]: engine room temperature controller external setpoint run*) (*OldName:Wex_RTMREG; Cycle:5;*)
		tiPurgeTimeMax : TIME; (*PARA [12296]: purge time maximum (room vent. before start without feedback)*) (*OldName:PurgeTimeMax; Cycle:5;*)
		bPurgecycle_Active : BOOL; (*PARA [12256]: purge cycle enable *) (*OldName:bPurgecycle; Cycle:5;*)
		bOutAirER_Lou1_visible : BOOL; (*PARA [12254]: outlet air engine room louver 1 visible*) (*OldName:bAirOutLou; Cycle:5;*)
		bInAirER_Lou2_visible : BOOL; (*PARA [12252]: intake air engine room louver 2 visible*) (*OldName:bAirInLou2; Cycle:5;*)
		bInAirER_Lou1_visible : BOOL; (*PARA [12251]: intake air engine room louver 1 visible*) (*OldName:bAirInLou1; Cycle:5;*)
		bInAirER_Fan2_visible : BOOL; (*PARA [12250]: intake air engine room fan 2 visible*) (*OldName:bAirInVent2; Cycle:5;*)
		bInAirER_Fan1_visible : BOOL; (*PARA [12249]: intake air engine room fan 1 visible*) (*OldName:bAirInVent1; Cycle:5;*)
		bInAirER_Fan_FU : BOOL; (*PARA [12248]: intake air engine room fan with frequency controller*) (*OldName:bAirInVentF; Cycle:5;*)
		rT_InAirER_LimHi : REAL; (*PARA [12274]: intake air engine room temperature limit high*) (*OldName:ssIATempMax; Cycle:5;*)
		rT_AirER_HyHi4 : REAL; (*PARA [12265]: air engine room temperature limit high 4 hysteresis*) (*OldName:HY_RTM_4; Cycle:5;*)
		rT_AirER_HyHi3 : REAL; (*PARA [12264]: air engine room temperature limit high 3 hysteresis*) (*OldName:HY_RTM_3; Cycle:5;*)
		rT_AirER_HyHi2 : REAL; (*PARA [12263]: air engine room temperature limit high 2 hysteresis*) (*OldName:HY_RTM_2; Cycle:5;*)
		rT_AirER_HyHi1 : REAL; (*PARA [12262]: air engine room temperature limit high 1 hysteresis*) (*OldName:HY_RTM_1; Cycle:5;*)
		rT_AirER_HyHi : REAL; (*PARA [12261]: air engine room temperature limit high hysteresis*) (*OldName:HY_RTM; Cycle:5;*)
		rT_Fan_InAirER_HyHi : REAL; (*PARA [12273]: intake air engine room temperature limit demand fan hysteresis*) (*OldName:HY_ASLT_V; Cycle:5;*)
		rT_Lou_InAirER_HyHi : REAL; (*PARA [12277]: intake air engine room temperature limit demand open louvers hysteresis*) (*OldName:HY_ASLT_J; Cycle:5;*)
		rT_AirER_LimHi4 : REAL; (*PARA [12270]: air engine room temperature limit high 4*) (*OldName:GW_RTM_4; Cycle:5;*)
		rT_AirER_LimHi3 : REAL; (*PARA [12269]: air engine room temperature limit high 3*) (*OldName:GW_RTM_3; Cycle:5;*)
		rT_AirER_LimHi2 : REAL; (*PARA [12268]: air engine room temperature limit high 2*) (*OldName:GW_RTM_2; Cycle:5;*)
		rT_AirER_LimHi1 : REAL; (*PARA [12267]: air engine room temperature limit high 1*) (*OldName:GW_RTM_1; Cycle:5;*)
		rT_AirER_LimHi : REAL; (*PARA [12266]: air engine room temperature limit high *) (*OldName:GW_RTM; Cycle:5;*)
		rT_InAirER_LimHi_Fan : REAL; (*PARA [12275]: intake air engine room temperature limit demand fan *) (*OldName:GW_ASLT_V; Cycle:5;*)
		rT_InAirER_LimHi_Lou : REAL; (*PARA [12276]: intake air engine room temperature limit demand open louvers *) (*OldName:GW_ASLT_J; Cycle:5;*)
		bPred_T_InAirER_Active : BOOL; (*PARA [12255]: intake air engine room temperature power reduction active*) (*OldName:bIATempRed; Cycle:5;*)
		rT_Pred_InAirER_Start : REAL; (*PARA [12280]: intake air engine room temperature power reduction start [°C]*) (*OldName:ssIATempRedStart; Cycle:5;*)
		rT_Pred_InAirER_Rate : REAL; (*PARA [12278]: intake air engine room temperature power reduction rate [%Pnom/°C]*) (*OldName:ssIATempRedRate; Cycle:5;*)
		rT_Pred_InAirER_Start2 : REAL; (*PARA [12281]: intake air engine room temperature power reduction start 2 [°C]*) (*OldName:ssIATempRedStart2; Cycle:5;*)
		rT_Pred_InAirER_Rate2 : REAL; (*PARA [12279]: intake air engine room temperature power reduction rate 2 [%Pnom/°C]*) (*OldName:ssIATempRedRate2; Cycle:5;*)
		bT_AirER_Active : BOOL; (*PARA [12257]: intake air engine room temperature measuremnet enable *) (*OldName:bRoomTemp; Cycle:5;*)
		bT_InAirER_Active : BOOL; (*PARA [12258]: intake air engine room temperature measurement enable *) (*OldName:bIATempAct; Cycle:5;*)
		rP_Dev_LimHi : REAL; (*PARA [12260]: power deviation (actual value/reduced set value) limit high [%/P_nom]*) (*OldName:Z_GW_PDIFF; Cycle:5;*)
		tiP_Dev_LimHi_Delay : TIME; (*PARA [12295]: power deviation (actual value/reduced set value) high, delay time*) (*OldName:T99; Cycle:5;*)
		bERV_AirFlowMon_Active : BOOL; (*PARA [12247]: eng.room vent.air flow monitoring active*) (*OldName:bERV_AirFlowMon_Active; Cycle:5;*)
		rN_EngStart_HyHi : REAL; (*PARA [11295]: speed engine start limit high hysteresis *) (*OldName:HY_DREHZ; Cycle:5*)
		rN_EngStart_LimHi : REAL; (*PARA [11296]: speed engine start limit high *) (*OldName:GW_DREHZ; Cycle:5*)
		bCtr_InlLou : BOOL; (*PARA [13068]: air inlet louver controller enable*) (*OldName:newPv; Cycle:5;*) (*STM*)
		bCtr_OutlLou_RT : BOOL; (*PARA [13078]: air outlet louver controller for room temperature enable*) (*OldName:newPv; Cycle:5;*) (*STM 2*)
		bCtr_OutlLou_RDP : BOOL; (*PARA [13262]: air outlet louver controller for room differential pressure enable*) (*OldName:newPv; Cycle:5;*) (*STM 2*)
		bCtr_CircLou : BOOL; (*PARA [13116]: air circulation louver controller enable*) (*OldName:newPv; Cycle:5;*) (*STM*)
		bPos_InlLou1_Active : BOOL; (*PARA [13069]: air inlet louver 1 position measuring enable*) (*OldName:newPv; Cycle:5;*) (*STM*)
		bPos_InlLou2_Active : BOOL; (*PARA [13072]: air inlet louver 2 position measuring enable*) (*OldName:newPv; Cycle:5;*) (*STM*)
		bPos_OutlLou1_Active : BOOL; (*PARA [13079]: air outlet louver 1 position measuring enable*) (*OldName:newPv; Cycle:5;*) (*STM*)
		bPos_OutlLou2_Active : BOOL; (*PARA [13084]: air outlet louver 2 position measuring enable*) (*OldName:newPv; Cycle:5;*) (*STM*)
		bPos_CircLou1_Active : BOOL; (*PARA [13138]: air circulation louver 1 position measuring enable*) (*OldName:newPv; Cycle:5;*) (*STM*)
		bPos_CircLou2_Active : BOOL; (*PARA [13143]: air circulation louver 2 position measuring enable*) (*OldName:newPv; Cycle:5;*) (*STM*)
		bInlVent_Ctr_InlLou_Active : BOOL; (*PARA [13075]: room ventilation with controllable inlet louver active*) (*OldName:newPv; Cycle:5;*) (*STM*)
		bOutlVent_Ctr_OutlLou_Active : BOOL; (*PARA [13088]: room ventilation with controllable out louver active*) (*OldName:newPv; Cycle:5;*) (*STM*)
		rPosLim_InlLou_Rel_FC_ER : REAL; (*PARA [13076]: minimal air inlet louver(s) position for release frequency converter room ventilation (FG_FU)*) (*OldName:newPv; Cycle:5;*) (*STM*)
		rPosLim_InlLou_Rel_FC_ER_Hy : REAL; (*PARA [13077]: minimal air inlet louver(s) position for release frequency converter room ventilation (FG_FU) hysteresis*) (*OldName:newPv; Cycle:5;*) (*STM*)
		tCtr_InlLou : _tGeACtrPara; (*Para controller air inlet louvers (for engine room temperature)*) (*OldName:newPv; Cycle:5;*) (*STM*)
		tCtr_OutlLou_RT : _tGeACtrPara; (*Para controller air outlet louvers (for engine room temperature)*) (*OldName:newPv; Cycle:5;*) (*STM 2*)
		tCtr_OutlLou_RDP : _tGeACtrPara; (*Para controller air outlet louvers (for engine room diffential pressure)*) (*OldName:newPv; Cycle:5;*) (*STM 2*)
		tCtr_CircLou : _tGeACtrPara; (*Para controller air circulation louvers (for engine intake air temperature)*) (*OldName:newPv; Cycle:5;*) (*STM*)
		bPrDiff_ER_Active : BOOL; (*PARA [13085]: engine room difference pressure enable*) (*OldName:newPv; Cycle:5;*) (*STM 2*)
		rPosLim_OutlLou_Rel_FC_ER : REAL; (*PARA [13089]: minimal air outlet louver(s) position for release frequency converter room ventilation (FG_FU)*) (*OldName:newPv; Cycle:5;*) (*STM*)
		rPosLim_OutlLou_Rel_FC_ER_Hy : REAL; (*PARA [13090]: minimal air outlet louver(s) position for release frequency converter room ventilation (FG_FU) hysteresis*) (*OldName:newPv; Cycle:5;*) (*STM*)
		rPrDiff_ER_Lim_High : REAL; (*PARA [13091]: limit high engine room differece pressure*) (*OldName:newPv; Cycle:5;*) (*STM 2*)
		rPrDiff_ER_Lim_High_Hy : REAL; (*PARA [13092]: limit high engine room difference pressure hysteresis*) (*OldName:newPv; Cycle:5;*) (*STM 2*)
		rPrDiff_ER_Lim_Low : REAL; (*PARA [13093]: limit low engine room differece pressure*) (*OldName:newPv; Cycle:5;*) (*STM 2*)
		rPrDiff_ER_Lim_Low_Hy : REAL; (*PARA [13094]: limit low engine room difference pressure hysteresis*) (*OldName:newPv; Cycle:5;*) (*STM 2*)
		rT_InAirER_Rel_CircOp : REAL; (*PARA [13144]: limit low engine intake air temperature for circulating operation release*) (*OldName:newPv; Cycle:5;*) (*STM*)
		rT_InAirER_Rel_CircOp_Hy : REAL; (*PARA [13145]: limit low engine intake air temperature for circulating operation release hysteresis*) (*OldName:newPv; Cycle:5;*) (*STM*)
		iTypeCtr_InlLou_ERV : INT; (*PARA [13817]: type control inlet louver(s)*) (*OldName:newPv; Cycle:5;*)
		iTypeCtr_OutlLou_ERV : INT; (*PARA [13818]: type control outlet louver(s)*) (*OldName:newPv; Cycle:5;*)
		iTypeFeedback_InlLou_ERV : INT; (*PARA [13819]: type feedback inlet louver(s)*) (*OldName:newPv; Cycle:5;*)
		iTypeFeedback_OutlLou_ERV : INT; (*PARA [13820]: type feedback outlet louver(s)*) (*OldName:newPv; Cycle:5;*)
		rPosLim_InlLou_Rel_ERV : REAL; (*PARA [13821]: minimal air inlet louver(s) position for release frequency converter room ventilation (FG_FU)*) (*OldName:newPv; Cycle:5;*)
		rPosLim_InlLou_Rel_ERV_Hy : REAL; (*PARA [13822]: minimal air inlet louver(s) position for release frequency converter room ventilation (FG_FU) hysteresis*) (*OldName:newPv; Cycle:5;*)
		rPosLim_OutlLou_Rel_ERV : REAL; (*PARA [13823]: minimal air outlet louver(s) position for release frequency converter room ventilation (FG_FU)*) (*OldName:newPv; Cycle:5;*)
		rPosLim_OutlLou_Rel_ERV_Hy : REAL; (*PARA [13824]: minimal air outlet louver(s) position for release frequency converter room ventilation (FG_FU) hysteresis*) (*OldName:newPv; Cycle:5;*)
		tCtr_OutlVE_RT : _tGeACtrPara; (*Para controller air outlet ventilation (for engine room temperature)*) (*OldName:newPv; Cycle:5;*) (*STM 2*)
		bCtr_OutlVE_RT : BOOL; (*PARA [13540]: air outlet ventilation controller for room temperature enable*)
		tCtr_OutlVE_RDP : _tGeACtrPara; (*Para controller air outlet ventilation (for engine room differential pressure)*) (*OldName:newPv; Cycle:5;*) (*STM 2*)
		bCtr_OutlVE_RDP : BOOL; (*PARA [13563]: air outlet ventilation controller for room differential pressure enable*)
		rVent_SpeedDif : REAL; (*PARA [13586]: speed difference [%] air inlet ventilation to air outlet ventilation in case of MSF engine room differential pressure*)
		bOutAirER_Fan_FU : BOOL; (*PARA [13541]: outlet air engine room fan with frequency controller*) (*OldName:newPv; Cycle:5;*)
		bCtr_RDP_OutlVE_Dep_InlVent : BOOL; (*PARA [13846]: activation ctr room differential pressure with outlet ventilation depending on ctr-signal inlet ventilation*)
		rScal_CtrInlVentER_Set_Min : REAL; (*PARA [13848]: minimal ctr-signal (speed-setpoint %) for room temperature-ctr inlet ventilation*)
		rScal_CtrInlVentER_Set_Max : REAL; (*PARA [13849]: maximal ctr-signal (speed-setpoint %) for room temperature-ctr inlet ventilation*)
		rScal_OffSetMin_CtrOutlVent : REAL; (*PARA [13850]: minimal offset (speed-setpoint %) for ctr outlet ventilation depending on ctr-signal inlet ventilation*)
		rScal_OffSetMax_CtrOutlVent : REAL; (*PARA [13851]: maximal offset (speed-setpoint %) for ctr outlet ventilation depending on ctr-signal inlet ventilation*)
		bCtr_RDP_OutlVE_Dep_EngP : BOOL; (*PARA [13847]: activation ctr room differential pressure with outlet ventilation depending on actual engine power*)
		rScal_PminEl : REAL; (*PARA [13852]: minimal engine power (%)  for load-related outlet ventilation control*)
		rScal_PmaxEl : REAL; (*PARA [13853]: maximal engine power (%)  for load-related outlet ventilation control*)
		rScal_OffSetMin_Pel : REAL; (*PARA [13854]: minimal offset (speed-setpoint %) for ctr outlet ventilation depending on acutal engine power*)
		rScal_OffSetMax_Pel : REAL; (*PARA [13855]: maximal offset (speed-setpoint %) for ctr outlet ventilation depending on ctr-signal inlet ventilation*)
		bFireProtFlap1_InlAir_visible : BOOL; (*PARA [13610]: fire protection flap 1 inlet air visible *) (*OldName:newPv; Cycle:5;*)
		bFireProtFlap2_InlAir_visible : BOOL; (*PARA [13611]: fire protection flap 2 inlet air visible *) (*OldName:newPv; Cycle:5;*)
		bFireProtFlap1_OutlAir_visible : BOOL; (*PARA [13612]: fire protection flap 1 outlet air visible *) (*OldName:newPv; Cycle:5;*)
		bFireProtFlap2_OutlAir_visible : BOOL; (*PARA [13613]: fire protection flap 2 outlet air visible *) (*OldName:newPv; Cycle:5;*)
		bBOP_ERVent_Act : BOOL; (*PARA [13836]: -Visu: Plant display room ventilation active*) (*OldName:newPv; Cycle:5;*)
		rT_ACP_AirER_sp : REAL; (*PARA [13987]: Active cooling program setpoint temperature engine room ventilation *)
		rT_AirER_LimWr : REAL; (*PARA [15064]: Room Temperature Warning*)
		bSafe_ERV_Cust_Active : BOOL; (*PARA [15188]: Customer room ventilation - Monitoring active*) (*SAFETY PLC; Cycle: 5;*) (*V04.25.00.00*)
	END_STRUCT;
END_TYPE
```

### module_VE.var
```iecst
VAR
	IN_VE : IN_Vent;
	OUT_VE : OUT_Vent;
	MM2VIS : MM2VIS_Struct;
	VIS2MM : VIS2MM_Struct;
	Para : Para_Vent;
	ParaFactoryDefault : Para_Vent := (0);
	pm : Para_Vent;
	xCtr_ER : GeACtr; (*controller engine room temperature*)
	tCtr_ER_In : _tGeACtrIn; (*controller engine room temperature*)
	tCtr_ER_Out : _tGeACtrOut; (*controller engine room temperature*)
	xCtr_InlLou : GeACtr; (*controller inlet louver (for engine room temperature)*) (*STM*)
	tCtr_InlLou_In : _tGeACtrIn; (*controller inlet louver (for engine room temperature)*) (*STM*)
	tCtr_InlLou_Out : _tGeACtrOut; (*controller inlet louver (for engine room temperature)*) (*STM*)
	xCtr_OutlLou_RT : GeACtr; (*controller outlet louver (for engine room temperature)*) (*STM 2*)
	tCtr_OutlLou_RT_In : _tGeACtrIn; (*controller outlet louver (for engine room temperature)*) (*STM 2*)
	tCtr_OutlLou_RT_Out : _tGeACtrOut; (*controller outlet louver (for engine room temperature)*) (*STM 2*)
	xCtr_OutlVE_RT : GeACtr; (*controller outlet ventilation (for engine room temperature)*) (*STM 2*)
	tCtr_OutlVE_RT_In : _tGeACtrIn; (*controller outlet ventilation (for engine room temperature)*) (*STM 2*)
	tCtr_OutlVE_RT_Out : _tGeACtrOut; (*controller outlet ventilation (for engine room temperature)*) (*STM 2*)
	xCtr_OutlVE_RDP : GeACtr; (*controller outlet ventilation (for engine room differential pressure)*) (*STM 2*)
	tCtr_OutlVE_RDP_In : _tGeACtrIn; (*controller outlet ventilation (for engine room differential pressure)*) (*STM 2*)
	tCtr_OutlVE_RDP_Out : _tGeACtrOut; (*controller outlet ventilation (for engine room differential pressure)*) (*STM 2*)
	xCtr_OutlLou_RDP : GeACtr; (*controller outlet louver (for engine room differential pressure)*) (*STM 2*)
	tCtr_OutlLou_RDP_In : _tGeACtrIn; (*controller outlet louver (for engine room differential pressure)*) (*STM 2*)
	tCtr_OutlLou_RDP_Out : _tGeACtrOut; (*controller outlet louver (for engine room differential pressure)*) (*STM 2*)
	xCtr_CircLou : GeACtr; (*controller circulation louver (for engine intake air temperature)*) (*STM*)
	tCtr_CircLou_In : _tGeACtrIn; (*controller circulation louver (for engine intake air temperature)*) (*STM*)
	tCtr_CircLou_Out : _tGeACtrOut; (*controller circulation louver (for engine intake air temperature)*) (*STM*)
	xOpMode : OpMode; (*engine operation mode*)
	xEngType : EngType; (*engine type*)
	bOMSS_Man : BOOL; (*engine operation mode selection*)
	bOMSS_Aut : BOOL; (*engine operation mode selection*)
	bOMSS_Test : BOOL; (*engine operation mode selection*)
	bOMSS_Scav : BOOL; (*engine operation mode selection*)
	bOMSS_MAT : BOOL; (*engine operation mode selection*)
	bGnlTrip : BOOL; (*general trip*)
	bCtrER_YFix : BOOL; (*demand engine room controller activation with fixed y*)
	bT_AirER_Hi_Wr : BOOL; (*air engine room temperature high *)
	bT_AirER_Hi : BOOL; (*air engine room temperature high *)
	bT_AirER_Hi1 : BOOL; (*air engine room temperature high *)
	bT_AirER_Hi2 : BOOL; (*air engine room temperature high *)
	bT_AirER_Hi3 : BOOL; (*air engine room temperature high *)
	bT_AirER_Hi4 : BOOL; (*air engine room temperature high *)
	bT_InAirER_LimHi_Lou : BOOL; (*intake air engine room temperature limit demand open louvers*)
	bT_InAirER_LimHi_Fan : BOOL; (*intake air engine room temperature limit demand fan*)
	ANF_LUE : BOOL; (*demand ventilation*)
	bGnlTrip1 : BOOL; (*general trip*)
	bGnlTrip2 : BOOL; (*general trip*)
	bGnlTrip3 : BOOL; (*general trip*)
	bGnlWarning : BOOL; (*general warning*)
	dmnd_purge : BOOL; (*demand purge cycle *)
	MS_LUE : BOOL; (*engine room ventilation signal failure summary*)
	FU_FIX : BOOL; (*freeze ER  frequency converter *)
	FG_FU : BOOL; (*release ER  frequency converter*)
	ZJAL2 : BOOL; (*inlet louver*)
	AJAL : BOOL; (*outlet louver*)
	ZJAL1 : BOOL; (*inlet louver*)
	RTM25 : BOOL; (*air engine room temperature high *)
	RTM30 : BOOL; (*air engine room temperature high *)
	RTM40 : BOOL; (*air engine room temperature high *)
	rT_AirER : REAL; (*air engine room temperature *)
	bNoInitDetected : BOOL := FALSE; (*always true, except 1cycle on init up*)
	Pos_InlLou1_OK : BOOL;
	Pos_OutlLou1_OK : BOOL;
	Pos_OutlLou2_OK : BOOL;
	Pos_InlLou2_OK : BOOL;
	M_DREHZ : BOOL; (* startup speed *)
	iValueInlLou : INT; (*value for inlet louvers case handling*)
	iValueOutlLou : INT; (*value for outlet louvers case handling*)
	bTON_DoorContact : BOOL := 0; (*Time delay door contact*)
	bERV_SafeCheck_CloseLou : BOOL; (*Safety plausibility checks close louver signal*)
	bERV_SafeCheck_OpenLou : BOOL; (*Safety plausibility checks open louver signal*)
END_VAR
```

### Program Logical/Ventilation/default_VE (IEC, version 4.07.0) - values

#### default_VECyclic.st
```iecst
(*******************************************************************************
default		value set

This code is confidential and proprietary to the INNIO Company.
It may not be used in any form, or reproduced in any manner,
without the express written permission of the INNIO Company.
Copyright, INNIO Company, 2019

Customized modifications: -
------------------------

History:
-------
V3.99.0		24.04.2012	lettenb.	new
V4.00.01	26.03.2014	lettenb.	tER_DoorClosed.Di added
V4.03.00	30.09.2015	lettenb.	tAuxV_Aux_ok and tAuxV_ModIf_ok added
V4.04.00	01.06.2016	Tinello		tDPr_InAirFiltERV_Hi added
V4.04.00    27.09.2016  Stary       added tER_InlAir_Ext_Err, tER_OutlAir_Ext_Err, tERV_InlAir_Op, tERV_OutlAir_Op
									moved default TRUE-settings for louvers to Vent_ER
V4.07.00    25.02.2019	Stary/lett. bAuxRel_FireProtFlaps: FireProtFlap feedback signals included in aux.release, safety case

Instructions for use:
--------------------
Outstandings:
------------
*******************************************************************************)
PROGRAM _CYCLIC

	(* default TRUE setting for not existing Di's *)
	IN_VE.tER_Ext_Err.Di			:=	IN_VE.tER_Ext_Err.Di			OR	NOT IN_VE.tER_Ext_Err.GoodQual;
	IN_VE.tER_InlAir_Ext_Err.Di		:=	IN_VE.tER_InlAir_Ext_Err.Di		OR	NOT IN_VE.tER_InlAir_Ext_Err.GoodQual;
	IN_VE.tER_OutlAir_Ext_Err.Di	:=	IN_VE.tER_OutlAir_Ext_Err.Di	OR	NOT IN_VE.tER_OutlAir_Ext_Err.GoodQual;
	IN_VE.tT_AirER_Ext_Hi.Di		:=	IN_VE.tT_AirER_Ext_Hi.Di		OR	NOT IN_VE.tT_AirER_Ext_Hi.GoodQual;
	IN_VE.tAuxV_Supply_Ok.Di		:=	IN_VE.tAuxV_Supply_Ok.Di		OR	NOT IN_VE.tAuxV_Supply_Ok.GoodQual;
	IN_VE.tAuxV_ModIf_ok.Di			:=	IN_VE.tAuxV_ModIf_ok.Di			OR	NOT IN_VE.tAuxV_ModIf_ok.GoodQual;				(*PJ*)
	IN_VE.tAuxV_Aux_ok.Di			:=	IN_VE.tAuxV_Aux_ok.Di			OR	NOT IN_VE.tAuxV_Aux_ok.GoodQual;			(*PJ*)
	IN_VE.tRel_ER_PurgeCycle.Di		:=	IN_VE.tRel_ER_PurgeCycle.Di		OR	NOT IN_VE.tRel_ER_PurgeCycle.GoodQual;
	IN_VE.tERV_Op.Di				:=	IN_VE.tERV_Op.Di				OR	NOT IN_VE.tERV_Op.GoodQual;
	IN_VE.tERV_InlAir_Op.Di         :=  IN_VE.tERV_InlAir_Op.Di         OR  NOT IN_VE.tERV_InlAir_Op.GoodQual;
	IN_VE.tERV_OutlAir_Op.Di        :=  IN_VE.tERV_OutlAir_Op.Di        OR  NOT IN_VE.tERV_OutlAir_Op.GoodQual;
	IN_VE.tER_DoorClosed.Di			:=	IN_VE.tER_DoorClosed.Di			OR	NOT IN_VE.tER_DoorClosed.GoodQual;
	IN_VE.tDPr_InAirFiltERV_Hi.Di 	:= 	IN_VE.tDPr_InAirFiltERV_Hi.Di 	OR	NOT IN_VE.tDPr_InAirFiltERV_Hi.GoodQual;	(* old: E_FILTER *)

	IN_VE.tFireProtFlap1_InlAir_Opened.Di  := IN_VE.tFireProtFlap1_InlAir_Opened.Di  OR NOT IN_VE.tFireProtFlap1_InlAir_Opened.GoodQual;
	IN_VE.tFireProtFlap2_InlAir_Opened.Di  := IN_VE.tFireProtFlap2_InlAir_Opened.Di  OR NOT IN_VE.tFireProtFlap2_InlAir_Opened.GoodQual;
	IN_VE.tFireProtFlap1_OutlAir_Opened.Di := IN_VE.tFireProtFlap1_OutlAir_Opened.Di OR NOT IN_VE.tFireProtFlap1_OutlAir_Opened.GoodQual;
	IN_VE.tFireProtFlap2_OutlAir_Opened.Di := IN_VE.tFireProtFlap2_OutlAir_Opened.Di OR NOT IN_VE.tFireProtFlap2_OutlAir_Opened.GoodQual;
	IN_VE.tFireProtFlap1_InlAir_Closed.Di  := IN_VE.tFireProtFlap1_InlAir_Closed.Di  OR NOT IN_VE.tFireProtFlap1_InlAir_Closed.GoodQual;
	IN_VE.tFireProtFlap2_InlAir_Closed.Di  := IN_VE.tFireProtFlap2_InlAir_Closed.Di  OR NOT IN_VE.tFireProtFlap2_InlAir_Closed.GoodQual;
	IN_VE.tFireProtFlap1_OutlAir_Closed.Di := IN_VE.tFireProtFlap1_OutlAir_Closed.Di OR NOT IN_VE.tFireProtFlap1_OutlAir_Closed.GoodQual;
	IN_VE.tFireProtFlap2_OutlAir_Closed.Di := IN_VE.tFireProtFlap2_OutlAir_Closed.Di OR NOT IN_VE.tFireProtFlap2_OutlAir_Closed.GoodQual;

END_PROGRAM
```

### Program Logical/Ventilation/general_VE (IEC, version 4.05.0) - functions

#### general_VECyclic.st
```iecst
(*******************************************************************************
general			general functions

This code is confidential and proprietary to the INNIO Company.
It may not be used in any form, or reproduced in any manner,
without the express written permission of the INNIO Company.
Copyright, INNIO Company, 2019

Customized modifications: -
------------------------

History:
-------
V3.99.0	24.04.2012	lettenb.	new
V4.05.0 11.12.2017	lettenb.	check para setup added

Instructions for use:
--------------------
Outstandings:
------------
*******************************************************************************)
PROGRAM _CYCLIC

	(* check para setup *)
	IN_VE.tPB2MM.bParaSetupOk;
	Para.iEng_Motortype;    (* MIN= 208   MAX= 920    *)
	Para.rN_EngStart_LimHi; (* MIN= 50.0  MAX= 2200.0 *)

	(* engine type defnition *)
	xEngType.Motortype := INT_TO_UINT(Para.iEng_Motortype);
	xEngType();

	(* engine operating mode selection *)
	bOMSS_Man  := FALSE;
	bOMSS_Aut  := FALSE;
	bOMSS_Test := FALSE;
	bOMSS_Scav := FALSE;
	bOMSS_MAT  := FALSE;

	CASE IN_VE.iIdx_OMSS OF
	1:	bOMSS_Man  := TRUE;
		bOMSS_MAT  := TRUE;
	2:	bOMSS_Aut  := TRUE;
		bOMSS_MAT  := TRUE;
	3:	bOMSS_Test := TRUE;
		bOMSS_MAT  := TRUE;
	4:	bOMSS_Scav := TRUE;
	END_CASE;

	(* engine operating mode *)
	xOpMode(in:= IN_VE.iSt_OpMode);

	(*---------------------------------------------------------------------------*)
	(* start speed exceeded *)
	xGR_MAXR_DREHZ(In:= IN_VE.rN_EngAct, Gw:= Para.rN_EngStart_LimHi, Hy:= Para.rN_EngStart_HyHi);
	xTOF_M_DREHZ(IN:= xGR_MAXR_DREHZ.Q AND IN_VE.tPB2MM.bParaSetupOk, PT:= T#10s);
	M_DREHZ := xTOF_M_DREHZ.Q;

END_PROGRAM
```

#### general_VE.var
```iecst
VAR
	xGR_MAXR_DREHZ : GR_MAXR;
	xTOF_M_DREHZ : TOF;
END_VAR
```

### Program Logical/Ventilation/Vent_ER (IEC, version 4.25.0) - ventilation engine room
